FUNCTION_BLOCK FC_HeatingCurve_Test EXTENDS FB_TestSuite
VAR

END_VAR

TAmbNegative();
TAmbZero();
HeatingCurveZero();
HeatingCurveNegative();

METHOD HeatingCurveNegative // This method checks whether the heating curve can have a negative value
VAR
	HeatingCurveRes: Real;		//Actual value for Heating Curve
	ExpectedValue : REAL := -1;	//Expected value for Heating Curve
	fSlope: REAL := -1;				//Slope of Heating Curve
	fOffset: REAL := 35;				//Offset of Heating Curve

END_VAR
TEST('HeatingCurveNegative');
 
HeatingCurveRes := FC_HeatingCurve(fTempAmb := 36, fSlope, fOffset);
 
AssertEquals(Expected := ExpectedValue,
             Actual := HeatingCurveRes,
             Message := 'The calculation is not correct');
 
TEST_FINISHED();
END_METHOD

METHOD HeatingCurveZero // This method checks whether the heating curve can have zero as value
VAR
	HeatingCurveRes: REAL;		//Actual value for Heating Curve
	ExpectedValue : REAL := 0;  //Expected value for Heating Curve
	fSlope: REAL := -1;				//Slope of Heating Curve
	fOffset: REAL := 35;				//Offset of Heating Curve
//	fTempAmb: REAL

END_VAR
TEST('HeatingCurveZero');
 
HeatingCurveRes := FC_HeatingCurve(fTempAmb := 35, fSlope, fOffset);
 
AssertEquals(Expected := ExpectedValue,
             Actual := HeatingCurveRes,
             Message := 'The calculation is not correct');
 
TEST_FINISHED();
END_METHOD

METHOD TAmbNegative // This method checks whether negative ambient temperatures work properly
VAR
	HeatingCurveRes: REAL;		 //Actual value for Heating Curve
	ExpectedValue : REAL := 40;  //Expected value for Heating Curve
	fSlope: REAL := -1;				 //Slope of Heating Curve
	fOffset: REAL := 35;				 //Offset of Heating Curve
END_VAR
TEST('TAmbNegative');
 
HeatingCurveRes := FC_HeatingCurve(fTempAmb := -5, fSlope, fOffset);
 
AssertEquals(Expected := ExpectedValue,
             Actual := HeatingCurveRes,
             Message := 'The calculation is not correct');
 
TEST_FINISHED();
END_METHOD

METHOD TAmbZero // This method checks whether zero degrees as ambient temperature work properly
VAR
	HeatingCurveRes : REAL;		  //Actual value for Heating Curve
	ExpectedValue : REAL := 35;   //Expected value for Heating Curve
	fSlope: REAL := -1;				  //Slope of Heating Curve	
	fOffset: REAL := 35;				  //Offset of Heating Curve

END_VAR
TEST('TAmbZero');
 
HeatingCurveRes := FC_HeatingCurve(fTempAmb := 0, fSlope, fOffset);
 
AssertEquals(Expected := ExpectedValue,
             Actual := HeatingCurveRes,
             Message := 'The calculation is not correct');
 
TEST_FINISHED();
END_METHOD

END_FUNCTION_BLOCK

(* stored: Version 1.1.0.1, ProductVersion 3.1.4024.6
   POU FC_HeatingCurve_Test: Id {a0fbec08-aee2-4a09-ad8e-4fec6d3e55ea}, SpecialFunc None
   Method HeatingCurveNegative: Id {cd412f18-f4d4-4d52-80e4-b8e76a515e81}
   Method HeatingCurveZero: Id {424d22b1-3775-47c3-8b57-f71514e68337}
   Method TAmbNegative: Id {a9b84f90-43cf-4025-b7cf-c78c31734e9e}
   Method TAmbZero: Id {f01a7258-79a5-45f6-8cc2-c4fcb7f06c95} *)
